{attribute 'qualified_only'}
{attribute 'strict'}
TYPE EWPMaterial :
(
	black := 1,
	white := 2,
	metallic :=3,
	undetermined :=4,
	enum_member := 0
);
END_TYPE

(* stored: Version 1.1.0.1
   DUT EWPMaterial: Id {cfe01a5d-b723-43a5-be57-dab1b7b77498} *)
